// Mitsubishi GX Works2 project: 2023-05-18 #2 생산자동화기능사 3번   PLC: Q03UDV
// 생산자동화기능사

// global labels: Global1
VAR_GLOBAL
  PB1 AT X0 : BOOL;
  PB2 AT X1 : BOOL;
  정지 AT X2 : BOOL;
  공급후진 AT X3 : BOOL;
  공급전진 AT X4 : BOOL;
  가공후진 AT X5 : BOOL;
  가공전진 AT X6 : BOOL;
  송출후진 AT X7 : BOOL;
  송출전진 AT X8 : BOOL;
  배출후진 AT X9 : BOOL;
  배출전진 AT X0A : BOOL;
  매거진 AT X0B : BOOL;
  금속센서 AT X0F : BOOL;
  PB3 AT X0C : BOOL;
  적색 AT Y20 : BOOL;
  황색 AT Y21 : BOOL;
  녹색 AT Y22 : BOOL;
  공급1 AT Y23 : BOOL;
  공급2 AT Y24 : BOOL;
  가공 AT Y25 : BOOL;
  드릴 AT Y26 : BOOL;
  송출 AT Y27 : BOOL;
  배출 AT Y28 : BOOL;
  컨베이어 AT Y29 : BOOL;
END_VAR

PROGRAM 단속연속
VAR
  STATE : INT;
  MODE : INT;
  METAL : INT;
END_VAR
VAR CONSTANT
  단속 : INT;
  연속 : INT := 1;
  금속 : INT := 1;
  비금속 : INT := 2;
END_VAR
VAR
  점멸1 : ARRAY [0..3] OF BOOL;
  SWP : BOOL;
  점멸2 : ARRAY [0..3] OF BOOL;
  EMSTP : INT;
  컨베이어_1 : BOOL;
  드릴_1 : BOOL;
  녹색_1 : BOOL;
  황색_1 : BOOL;
  STATE_1 : INT;
END_VAR
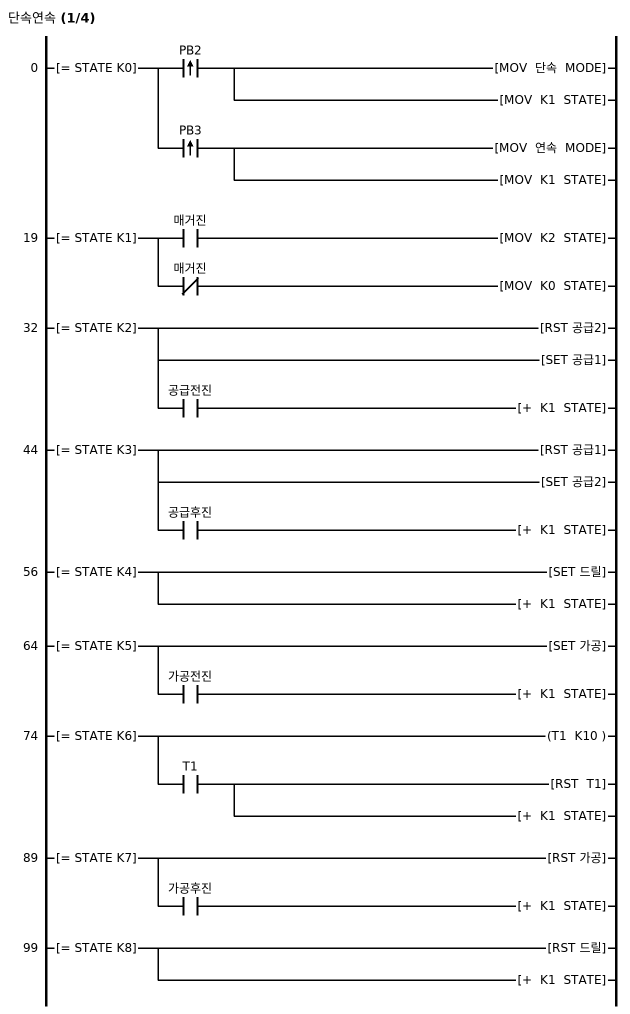
0     LD=     STATE K0
      MPS
      ANDP    PB2
      MOV     단속 MODE
      MOV     K1 STATE
      MPP
      ANDP    PB3
      MOV     연속 MODE
      MOV     K1 STATE
19    LD=     STATE K1
      MPS
      AND     매거진
      MOV     K2 STATE
      MPP
      ANI     매거진
      MOV     K0 STATE
32    LD=     STATE K2
      RST     공급2
      SET     공급1
      AND     공급전진
      +       K1 STATE
44    LD=     STATE K3
      RST     공급1
      SET     공급2
      AND     공급후진
      +       K1 STATE
56    LD=     STATE K4
      SET     드릴
      +       K1 STATE
64    LD=     STATE K5
      SET     가공
      AND     가공전진
      +       K1 STATE
74    LD=     STATE K6
      OUT     T1 K10
      AND     T1
      RST     T1
      +       K1 STATE
89    LD=     STATE K7
      RST     가공
      AND     가공후진
      +       K1 STATE
99    LD=     STATE K8
      RST     드릴
      +       K1 STATE
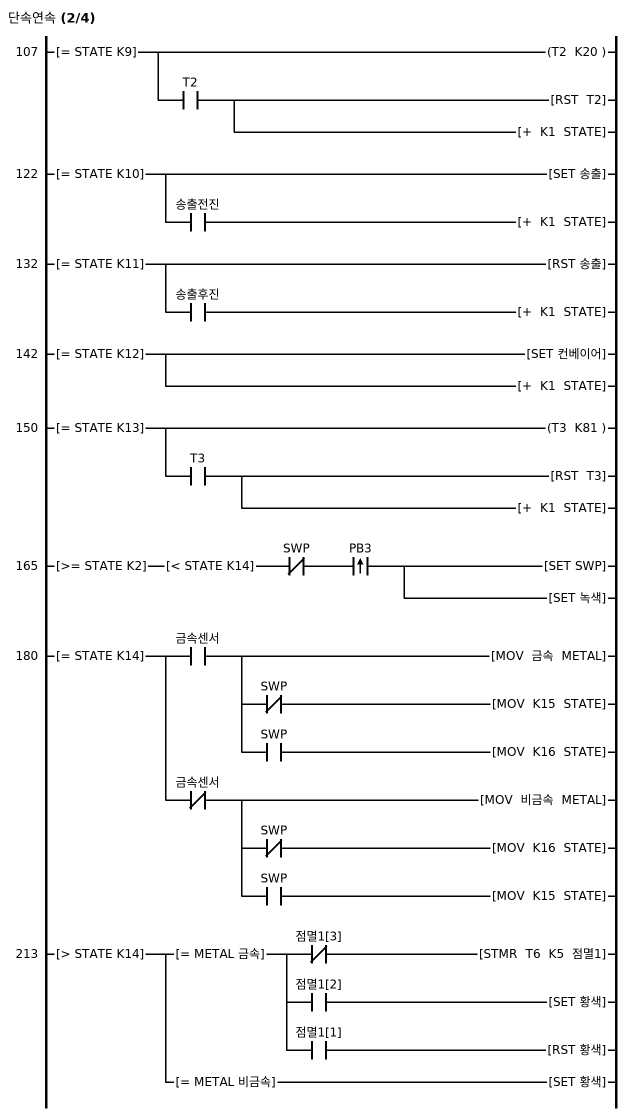
107   LD=     STATE K9
      OUT     T2 K20
      AND     T2
      RST     T2
      +       K1 STATE
122   LD=     STATE K10
      SET     송출
      AND     송출전진
      +       K1 STATE
132   LD=     STATE K11
      RST     송출
      AND     송출후진
      +       K1 STATE
142   LD=     STATE K12
      SET     컨베이어
      +       K1 STATE
150   LD=     STATE K13
      OUT     T3 K81
      AND     T3
      RST     T3
      +       K1 STATE
165   LD>=    STATE K2
      AND<    STATE K14
      ANI     SWP
      ANDP    PB3
      SET     SWP
      SET     녹색
180   LD=     STATE K14
      MPS
      AND     금속센서
      MOV     금속 METAL
      MPS
      ANI     SWP
      MOV     K15 STATE
      MPP
      AND     SWP
      MOV     K16 STATE
      MPP
      ANI     금속센서
      MOV     비금속 METAL
      MPS
      ANI     SWP
      MOV     K16 STATE
      MPP
      AND     SWP
      MOV     K15 STATE
213   LD>     STATE K14
      MPS
      AND=    METAL 금속
      MPS
      ANI     점멸1[3]
      STMR    T6 K5 점멸1
      MRD
      AND     점멸1[2]
      SET     황색
      MPP
      AND     점멸1[1]
      RST     황색
      MPP
      AND=    METAL 비금속
      SET     황색
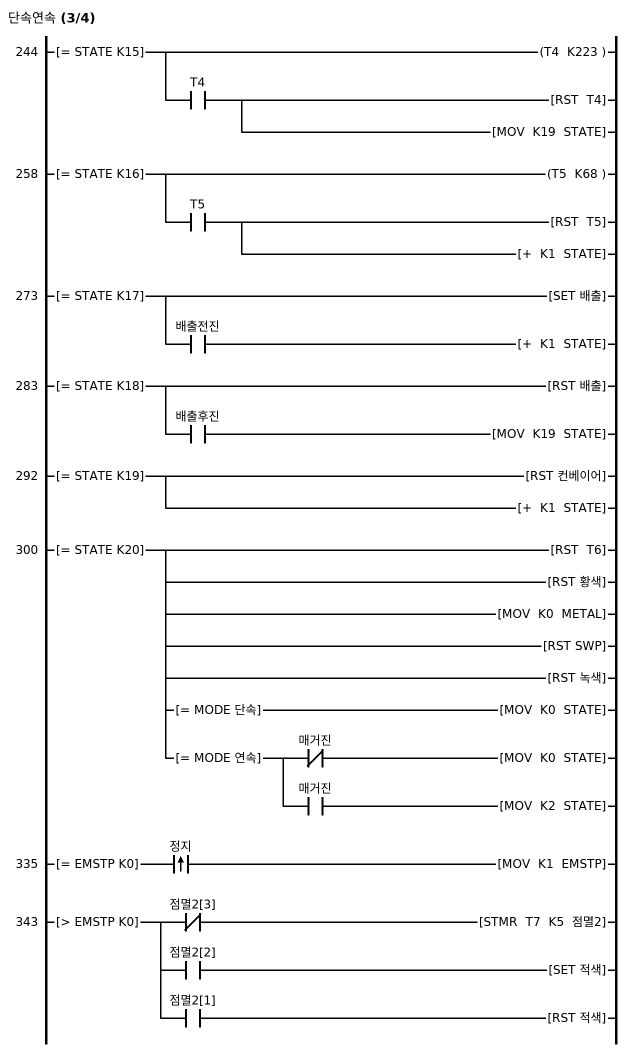
244   LD=     STATE K15
      OUT     T4 K223
      AND     T4
      RST     T4
      MOV     K19 STATE
258   LD=     STATE K16
      OUT     T5 K68
      AND     T5
      RST     T5
      +       K1 STATE
273   LD=     STATE K17
      SET     배출
      AND     배출전진
      +       K1 STATE
283   LD=     STATE K18
      RST     배출
      AND     배출후진
      MOV     K19 STATE
292   LD=     STATE K19
      RST     컨베이어
      +       K1 STATE
300   LD=     STATE K20
      RST     T6
      RST     황색
      MOV     K0 METAL
      RST     SWP
      RST     녹색
      MPS
      AND=    MODE 단속
      MOV     K0 STATE
      MPP
      AND=    MODE 연속
      MPS
      ANI     매거진
      MOV     K0 STATE
      MPP
      AND     매거진
      MOV     K2 STATE
335   LD=     EMSTP K0
      ANDP    정지
      MOV     K1 EMSTP
343   LD>     EMSTP K0
      MPS
      ANI     점멸2[3]
      STMR    T7 K5 점멸2
      MRD
      AND     점멸2[2]
      SET     적색
      MPP
      AND     점멸2[1]
      RST     적색
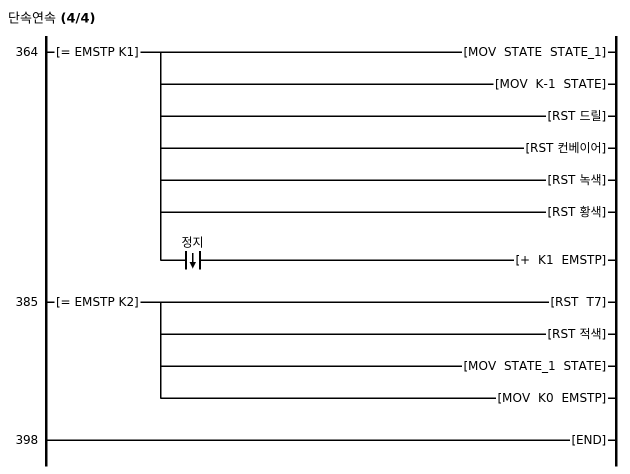
364   LD=     EMSTP K1
      MOV     STATE STATE_1
      MOV     K-1 STATE
      RST     드릴
      RST     컨베이어
      RST     녹색
      RST     황색
      ANDF    정지
      +       K1 EMSTP
385   LD=     EMSTP K2
      RST     T7
      RST     적색
      MOV     STATE_1 STATE
      MOV     K0 EMSTP
398   END
END_PROGRAM

PROGRAM 테스트
VAR
  STATE : INT;
END_VAR
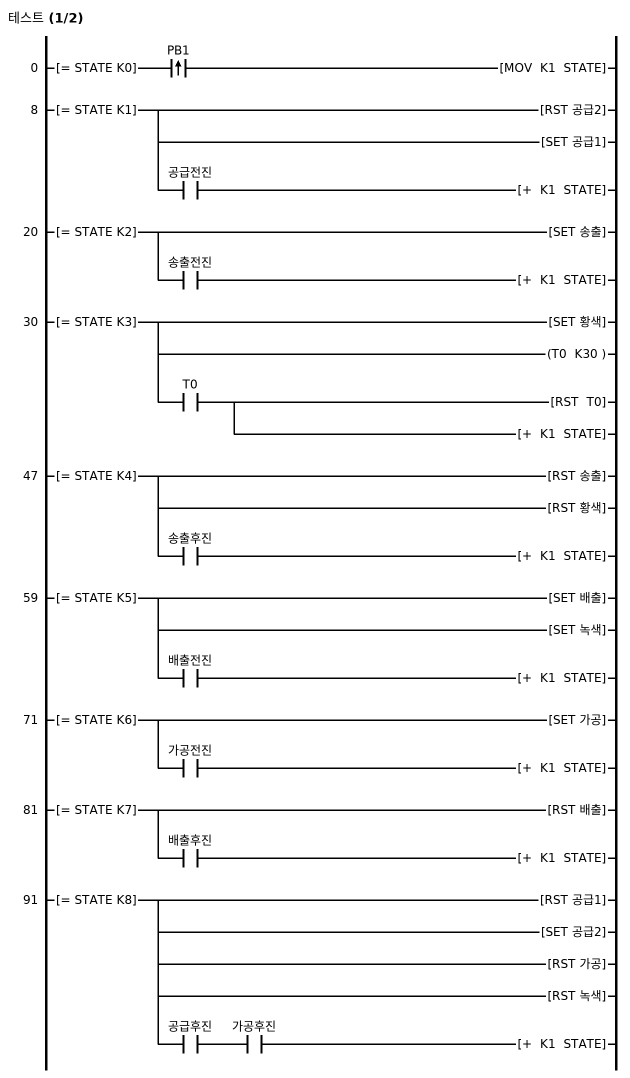
0     LD=     STATE K0
      ANDP    PB1
      MOV     K1 STATE
8     LD=     STATE K1
      RST     공급2
      SET     공급1
      AND     공급전진
      +       K1 STATE
20    LD=     STATE K2
      SET     송출
      AND     송출전진
      +       K1 STATE
30    LD=     STATE K3
      SET     황색
      OUT     T0 K30
      AND     T0
      RST     T0
      +       K1 STATE
47    LD=     STATE K4
      RST     송출
      RST     황색
      AND     송출후진
      +       K1 STATE
59    LD=     STATE K5
      SET     배출
      SET     녹색
      AND     배출전진
      +       K1 STATE
71    LD=     STATE K6
      SET     가공
      AND     가공전진
      +       K1 STATE
81    LD=     STATE K7
      RST     배출
      AND     배출후진
      +       K1 STATE
91    LD=     STATE K8
      RST     공급1
      SET     공급2
      RST     가공
      RST     녹색
      AND     공급후진
      AND     가공후진
      +       K1 STATE
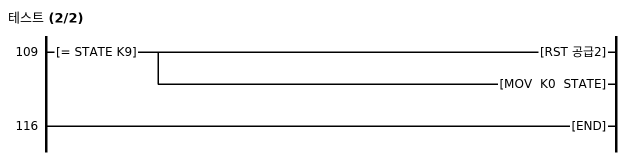
109   LD=     STATE K9
      RST     공급2
      MOV     K0 STATE
116   END
END_PROGRAM
